PROGRAM MAIN_obsolete
VAR
	robot1 : RobotLadder;
	robot2 : Robot;
	sensorBlock AT %I* : BIT8_ARRAY;
	//test : MDP5001_0_A368DC73;
END_VAR

robot1();
robot2();

END_PROGRAM

(* stored: Version 1.1.0.1, ProductVersion 3.1.4024.11
   POU MAIN_obsolete: Id {b128b248-c142-427a-98d0-25b88a13d8f0}, SpecialFunc None *)
